TYPE
   LongString : STRING(StringsParams.MAX_STRING_LENGTH);
END_TYPE // use StringsParams.MAX_STRING_LENGTH to adjust length

(* stored: Version 1.1.0.1, ProductVersion 3.1.4026.12
   DUT LongString: Id {f7b88719-a21a-07f5-306e-384a2fb17d37} *)
